TYPE ST_DIAGNOSTICCODE :
STRUCT
    eDiagnosticCodeType : E_DIAGNOSTICCODETYPE;
    nCode : UINT;
END_STRUCT
END_TYPE

(* stored: Version 1.1.0.1
   DUT ST_DIAGNOSTICCODE: Id {33760e3f-c166-46af-b1fa-3eff0f8bd21b} *)
